// This version uses the EL3161 and it's built in IIR filter
FUNCTION_BLOCK AnalogPrescaledSpeedCalculator IMPLEMENTS DemandedSpeedInterface; 
VAR_INPUT
	// Analog speed as 0-10v from PC Pin 13
	iAnalogSpeed AT %I*: INT;
END_VAR

METHOD GetSpeed : UINT
GetSpeed := TO_UINT(LIMIT(0, iAnalogSpeed, 24000))
END_METHOD

END_FUNCTION_BLOCK

(* stored: Version 1.1.0.1, ProductVersion 3.1.4022.16
   POU AnalogPrescaledSpeedCalculator: Id {331e867a-d9f4-4f14-8847-df60cde98080}, SpecialFunc None
   Method GetSpeed: Id {429766ce-4476-4106-9e75-9aee13cef53d} *)
